Yaskawa INFORM job: FAT.JBI

/JOB
//NAME FAT
///FOLDERNAME FOLDER001
//POS
///NPOS 0,0,0,0,0,0
//INST
///DATE 2023/07/11 09:16
///ATTR SC,RW,RJ
////FRAME ROBOT
NOP
CALL JOB:LEAVE_CAMERA
PAUSE
CALL JOB:CLEAN-R1
PAUSE
CALL JOB:MOTOTAC1
PAUSE
CALL JOB:GET_CAMERA
PAUSE
CALL JOB:SVETS
PAUSE
CALL JOB:R2-HOME
PAUSE
CALL JOB:R2-ST2-SAFE
PAUSE
CALL JOB:R2-ST1-SAFE
PAUSE
CALL JOB:SR-ARC-1
PAUSE
CALL JOB:TSYNC-R-TEST
PAUSE
CALL JOB:S1
END
